FUNCTION_BLOCK PICKER_RHMI_PROXY (* Communication Unit for Mirrored Picker HMI using a Socket *)
  (* Standard: 61499-2 *)
  (* Version 0.2, 2003-12-05, JHC, Rockwell Automation, Renamed from NEWCOMPFB. *)
  (* Version 0.1, 2002-01-08, JHC, Rockwell Automation, Added DLY FB as example. *)
  (* Version 0.0, 2000-05-27, JHC, Rockwell Automation *)
  (* Compiler header: package fb.rt.pnp;import fb.rt.net.*; *)
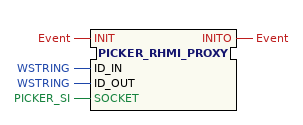
  EVENT_INPUT
    INIT; (* Initialization Request *)
  END_EVENT
  EVENT_OUTPUT
    INITO; (* Initialization Confirm *)
  END_EVENT
  VAR_INPUT
    ID_IN : WSTRING;
    ID_OUT : WSTRING;
  END_VAR
  SOCKETS
    SOCKET : PICKER_SI;
  END_SOCKETS
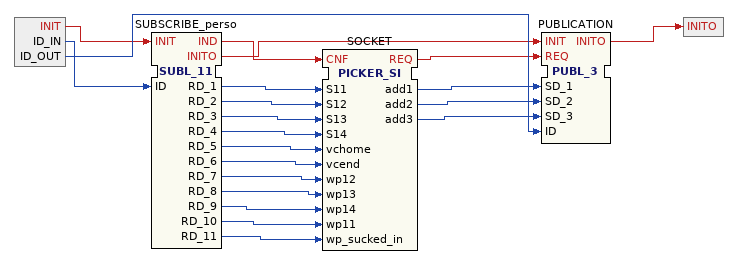
  FBS
    SUBSCRIBE_perso : SUBL_11;
    PUBLICATION : PUBL_3;
  END_FBS
  EVENT_CONNECTIONS
    INIT TO SUBSCRIBE_perso.INIT;
    SUBSCRIBE_perso.IND TO SOCKET.CNF;
    SUBSCRIBE_perso.INITO TO PUBLICATION.INIT;
    SOCKET.REQ TO PUBLICATION.REQ;
    PUBLICATION.INITO TO INITO;
  END_CONNECTIONS
  DATA_CONNECTIONS
    SUBSCRIBE_perso.RD_1 TO SOCKET.S11;
    SUBSCRIBE_perso.RD_2 TO SOCKET.S12;
    SUBSCRIBE_perso.RD_3 TO SOCKET.S13;
    SUBSCRIBE_perso.RD_4 TO SOCKET.S14;
    SUBSCRIBE_perso.RD_5 TO SOCKET.vchome;
    SUBSCRIBE_perso.RD_6 TO SOCKET.vcend;
    SUBSCRIBE_perso.RD_7 TO SOCKET.wp12;
    SUBSCRIBE_perso.RD_8 TO SOCKET.wp13;
    SUBSCRIBE_perso.RD_9 TO SOCKET.wp14;
    SUBSCRIBE_perso.RD_10 TO SOCKET.wp11;
    SUBSCRIBE_perso.RD_11 TO SOCKET.wp_sucked_in;
    ID_IN TO SUBSCRIBE_perso.ID;
    SOCKET.add1 TO PUBLICATION.SD_1;
    SOCKET.add2 TO PUBLICATION.SD_2;
    SOCKET.add3 TO PUBLICATION.SD_3;
    ID_OUT TO PUBLICATION.ID;
  END_CONNECTIONS
END_FUNCTION_BLOCK
